{attribute 'call_after_init'}
FUNCTION_BLOCK FB_AmphosMRC_Test EXTENDS FB_TestSuite
VAR_INPUT
END_VAR
VAR_OUTPUT
END_VAR
VAR
END_VAR

ErrorTriggers();
ErrorGoesBackToNormal();
NoError();

METHOD ErrorGoesBackToNormal
VAR
	fbAmphosMRC : FB_AmphosMRC := F_AmphosMRC_Error();
END_VAR
TEST('ErrorGoesBackToNormal');

fbAmphosMRC(bMRC := TRUE);
AssertFalse(fbAmphosMRC.bError, 'Error did not go back to normal');

TEST_FINISHED();
END_METHOD

METHOD ErrorTriggers
VAR
	fbAmphosMRC : FB_AmphosMRC := F_AmphosMRC_Error();
END_VAR
TEST('ErrorTriggers');

AssertTrue(fbAmphosMRC.bError, 'Error did not trigger');

TEST_FINISHED();
END_METHOD

METHOD NoError
VAR
	fbAmphosMRC : FB_AmphosMRC;
END_VAR
TEST('NoError');

fbAmphosMRC(
	bAmphosOn := TRUE,
	bMRC := TRUE
);
AssertFalse(fbAmphosMRC.bError, 'Error falsely triggered');

TEST_FINISHED();
END_METHOD

END_FUNCTION_BLOCK

(* stored: Version 1.1.0.1, ProductVersion 3.1.4020.14
   POU FB_AmphosMRC_Test: Id {ca336742-d98a-4fb2-803e-441a8fd1baa5}, SpecialFunc None
   Method ErrorGoesBackToNormal: Id {b67d5987-969e-4b68-8d88-ccaa51f6b5c3}
   Method ErrorTriggers: Id {867246c5-7880-462a-95dd-229505324cdb}
   Method NoError: Id {def34857-00a5-41f4-a9cb-e6d0f0ab21ec} *)
